{attribute 'linkalways'} 
{attribute 'no_explicit_call' := 'This FB is a CLASS and must be accessed using methods or properties'}
{attribute 'enable_dynamic_creation'}
FUNCTION_BLOCK _ETcVnStructuringElementShape EXTENDS EnumDatatypeBase
VAR
	localData : ETcVnStructuringElementShape;
	activeData : REFERENCE TO ETcVnStructuringElementShape;
	enumBaseDatatype : _DINT(localData);
END_VAR

METHOD PRIVATE AddLocalEnumeration
VAR_INPUT
	Enumeration : T_MAXSTRING;
	Value : ETcVnStructuringElementShape;
END_VAR
AddEnumeration(Enumeration, Value);
END_METHOD

PROPERTY PUBLIC Address : PVOID
GET
Address := ADR(activeData);
END_GET
END_PROPERTY

METHOD PUBLIC ClearReference
VAR_INPUT
END_VAR
activeData REF= localData;
SetBaseDatatypeReference();
END_METHOD

METHOD PUBLIC Clone : I_Datatype
VAR
    pClone : POINTER TO _ETcVnStructuringElementShape;
END_VAR
pClone := __NEW(_ETcVnStructuringElementShape(InitialValue := Value));
Clone := pClone^;
END_METHOD

METHOD FB_init : BOOL
VAR_INPUT
	bInitRetains : BOOL; // if TRUE, the retain variables are initialized (warm start / cold start)
	bInCopyCode : BOOL;  // if TRUE, the instance afterwards gets moved into the copy code (online change)
	InitialValue : ETcVnStructuringElementShape;
END_VAR
localData := InitialValue;
AddBaseDatatype(enumBaseDatatype);
ClearReference();

AddLocalEnumeration('TCVN_SES_RECTANGLE', ETcVnStructuringElementShape.TCVN_SES_RECTANGLE);
AddLocalEnumeration('TCVN_SES_CROSS', ETcVnStructuringElementShape.TCVN_SES_CROSS);
AddLocalEnumeration('TCVN_SES_ELLIPSE', ETcVnStructuringElementShape.TCVN_SES_ELLIPSE);
END_METHOD

PROPERTY PUBLIC Identifier : T_MAXSTRING
GET
Identifier := 'ETcVnStructuringElementShape';
END_GET
END_PROPERTY

METHOD IsEnumeratorValueEqual : BOOL
VAR_INPUT
	Enumerator : I_KeyValueForwardEnumerator;
END_VAR
VAR
	storedValue : ETcVnStructuringElementShape;
END_VAR
IF NOT Enumerator.TryGet(storedValue) THEN
	RETURN;
END_IF

IsEnumeratorValueEqual := storedValue = activeData;
END_METHOD

METHOD PUBLIC MakeReferenceTo
VAR_INPUT
	ReferenceTarget : REFERENCE TO ETcVnStructuringElementShape;
END_VAR
activeData REF= ReferenceTarget;
SetBaseDatatypeReference();
END_METHOD

METHOD PROTECTED SetBaseDatatypeReference
VAR_INPUT
END_VAR
enumBaseDatatype.MakeReferenceTo(activeData);
END_METHOD

PROPERTY PUBLIC Size : UDINT
GET
Size := SIZEOF(activeData);
END_GET
END_PROPERTY

METHOD TryMakeReferenceTo : BOOL
VAR_INPUT
	Target : I_Datatype;
END_VAR
VAR
	targetAsEnum : I_EnumDatatype;
	pTargetData : POINTER TO ETcVnStructuringElementShape;
END_VAR
IF NOT Target.TryResolveAsEnumDatatype(targetAsEnum) THEN
	RETURN;
END_IF

IF targetAsEnum.Identifier <> Identifier THEN
	RETURN;
END_IF

pTargetData := Target.Address;
activeData REF= pTargetData^;
SetBaseDatatypeReference();
TryMakeReferenceTo := TRUE;
END_METHOD

PROPERTY PUBLIC Value : ETcVnStructuringElementShape
GET
Value := activeData;
END_GET
SET
activeData := Value;
END_SET
END_PROPERTY

END_FUNCTION_BLOCK

(* stored: Version 1.1.0.1, ProductVersion 3.1.4024.12
   POU _ETcVnStructuringElementShape: Id {0279b147-0707-4641-a762-73a7bd98fbd3}, SpecialFunc None
   Folder Constructor: Id {2bc391e8-2925-4e68-9689-dfda400b9833}
   Folder Private: Id {512bab00-2dd0-4e7f-9c84-dc4be0a67e01}
   Folder Protected: Id {4eb8c8e2-e55d-41c7-a655-ee1c1ee27a73}
   Method AddLocalEnumeration: Id {c600d4c8-7802-4c7f-a86e-ee4179457d74}
   Property Address: Id {f2ed541e-8ec4-48ea-840f-e31726edc52f}
   Get Get: Id {eadb78d7-4aa8-4296-b050-592e19d6ef77}
   Method ClearReference: Id {70bc4222-97da-40ae-83d2-b3ef611f7603}
   Method Clone: Id {e522e208-3bf9-47e7-b113-b9a0543420ac}
   Method FB_init: Id {bcbd283d-c6ee-4161-b976-ad7fdd64c990}
   Property Identifier: Id {864171f6-d26d-4992-8c3a-cf7b5a2afe30}
   Get Get: Id {eb4d41a0-8cd9-478f-8497-15f53f50bd9e}
   Method IsEnumeratorValueEqual: Id {39a83c23-5319-4f24-a218-165c7deaa6f6}
   Method MakeReferenceTo: Id {c803190d-80d7-4cdf-902f-3793a21b55da}
   Method SetBaseDatatypeReference: Id {d7a405bb-b1bd-4c9e-93e0-a3eecf0bd41c}
   Property Size: Id {154f606c-2fde-4119-859d-23d36ca0fce2}
   Get Get: Id {e417a630-8ac1-4df6-8cc9-7fa8990d9879}
   Method TryMakeReferenceTo: Id {e826bd44-9d95-4311-b2b0-dfb18b5acd20}
   Property Value: Id {1b24572d-e7ab-4025-a071-d0ae9a6d76f4}
   Get Get: Id {e1c4db63-9812-4071-b68a-c2e04c430bbc}
   Set Set: Id {cb1147d0-35c3-41d1-ad83-02b97bbb2756} *)
